KUKA KRL program: BrakeTestSelfTest.src, BrakeTestSelfTest.dat

--- BrakeTestSelfTest.src ---
&ACCESS RVO
&REL 1
&PARAM EDITMASK = *
&PARAM TEMPLATE = C:\KRC\Roboter\Template\ExpertVorgabe
DEF BrakeTestSelfTest( )
Int Ret
Int IntArray[3]
Real RealArray[1]

MsgQuit("AcknowledgeToPerformSelfTest", brakeTestMdbName[])

; Bei der naechsten Test-Durchfuehrung das Ansprechverhalten
; einer Bremse oder aller Bremsen vorwählen
IntArray[1] = simulateBrakeVel
IntArray[2] = simulateBrakeTorque
IntArray[3] = simulateBrakeIndex
Ret = MD_CMD(brakeTestDevName[], "TRIGGER_SELF_TEST", IntArray[], RealArray[])

; Test-Anforderung erzwingen
MD_SETSTATE(brakeTestDevName[], #INITIALIZED)

; Test-Durchfuehrung
BrakeTestReq()
END

--- BrakeTestSelfTest.dat ---
&ACCESS RVO
DEFDAT BrakeTestSelfTest PUBLIC

INT simulateBrakeVel    = 100
INT simulateBrakeTorque = 50
INT simulateBrakeIndex  = 2

ENDDAT
